# EPICS autosave request: ipApp/Db/Rigol_DS1000Z_settings.req
$(P)$(R)ReadStatusScan.SCAN
$(P)$(R)TrigMode
$(P)$(R)TrigSweep
$(P)$(R)TrigSource
$(P)$(R)TrigSlope
$(P)$(R)TrigLevel
$(P)$(R)TrigHoldoff
$(P)$(R)TrigNoiseReject
$(P)$(R)TimeMode
$(P)$(R)TimeScale
$(P)$(R)TimeOffset
